# EPICS substitutions: apps/amqApp/Db/hps-trigger-alarms.substitutions
file "db/hps-trigger-alarms.db" {
    pattern { RATE, MINRATE, MINCURRENT }
            { B_DAQ_HPS:VTP:rate:02, 500, 4 }
            { B_DAQ_HPS:VTP:rate:03, 500, 4 }
            { B_DAQ_HPS:VTP:rate:06, 500, 4 }
            { B_DAQ_HPS:VTP:rate:07, 500, 4 }
            { B_DAQ_HPS:TS:livetime, 60,  4 }
            { B_DAQ:STA:hps1:dataRate, 16, 40 }
            { B_DAQ:STA:hps2:dataRate, 16, 40 }
}
